FUNCTION_BLOCK FB_HMIManager EXTENDS FB_BaseGroupElement IMPLEMENTS ITF_HMIManager, ITF_HMIManagerConfigure
VAR
	(*	Inicjalizacja		*)
	bInitializeCycle			: BOOL;
	bInitDone					: BOOL;
	(*	Konfiguracja		*)
	itfHMIConfigure			: ITF_HMIConfigure;		//moduł konfiguracji
	(*	Menu główne	*)
	itfMainMenu				: ITF_HMIEMenu;
	iNumberOfButtonMainMenu	: INT;
	(*	Obsługa zmiany strony	*)
	arrChangePageSupport	: ARRAY [0..GVL_HMIEConstans.MAX_NUMBER_OF_BUTTON_IN_MENU] OF ITF_ChangePageSupport;
	(*	Dana wspólne dla całego systemu	*)
	refstData				: REFERENCE TO ST_HMIManager;
END_VAR

IF (NOT THIS^.bInitializeCycle) THEN
	THIS^.bInitializeCycle		:= TRUE;
	THIS^.bInitDone				:= THIS^.InitializeCycle ();
ELSIF (THIS^.bInitDone) THEN
	THIS^.ExecuteCycle ();
END_IF

(*			
	RafalOS
	Rafał Osajda		13.11.2025		TC 4024.66
	Dodawanie elementów wywoływane z konfiguracji 
*)
METHOD PUBLIC AddElementFromConfiguration : BOOL
VAR_INPUT
	itfElements		: ITF_BaseTopElement_HMI;
END_VAR
END_METHOD

(*			
	RafalOS
	Rafał Osajda		29.10.2025		TC 4024.66
	Dodawanie intefejsu konfiguracji
*)
METHOD PUBLIC AddModulConfigure : BOOL
VAR_INPUT
	fbHMIConfigure			: ITF_HMIConfigure;
END_VAR
THIS^.itfHMIConfigure		:= fbHMIConfigure;
END_METHOD

(*			
	RafalOS
	Rafał Osajda		10.11.2025		TC 4024.66
	Główna metoda sterujaca wyświetlaniem dsanych na HMI
*)
METHOD PUBLIC ExecuteCycle
(*
	(* Testowanie MenuGlownego	*)
THIS^.itfMainMenu.Testing ();

	(*	Aktualizacja zmiennych przy zmianie strony	*)
IF (THIS^.itfMainMenu.IsChangePage ()) THEN
	THIS^.refstData.iNUmberOfActivePage	:= THIS^.itfMainMenu.GetNumberOfActriveScreen ();
	
END_IF

	(*	Odświerzenia strrony 	*)
IF (THIS^.arrChangePageSupport [THIS^.refstData.iNUmberOfActivePage] <> 0) THEN
	THIS^.arrChangePageSupport [THIS^.refstData.iNUmberOfActivePage].PreparePage ();
	//wyczyszczenie po ramce 
	//przygotowanie ramki
END_IF
	(*	Skasowanie flagi zmiany strony	*)
THIS^.itfMainMenu.ResetChangePage ();
*)
END_METHOD

METHOD FB_init : BOOL
VAR_INPUT
	bInitRetains : BOOL; // if TRUE, the retain variables are initialized (warm start / cold start)
	bInCopyCode : BOOL;  // if TRUE, the instance afterwards gets moved into the copy code (online change)
END_VAR
THIS^.SetText (eLocation := E_BaseLocation.pl, wsDescription := "HMI Menadżer");
THIS^.SetText (eLocation := E_BaseLocation.en, wsDescription := "HMI Manager");
THIS^.SetText (eLocation := E_BaseLocation.de, wsDescription := "HMI Manager");
THIS^.SetName (stName := THIS^.GetTexts ());
END_METHOD

METHOD PRIVATE InitializeCycle : BOOL
VAR
	bResult					: BOOL;
	iI: INT;
END_VAR
bResult				:= TRUE;

bResult				:= bResult AND THIS^.itfHMIConfigure.Configure (fbHMIManager := THIS^);

InitializeCycle		:= bResult;
END_METHOD

METHOD PUBLIC SetActiveButtonMainMenuFromConfiguration : BOOL
VAR_INPUT
	iButton			: INT;	//numer przycisku od 0
	bValue			: BOOL;	//true aktywny może być tylko jeden w menu
END_VAR
THIS^.itfMainMenu.SetActiveButton (iButton := iButton, bIN := bValue);
END_METHOD

METHOD PUBLIC SetEnableButtonMainMenuFromConfiguration : BOOL
VAR_INPUT
	iButton			: INT;	//numer przycisku od 0
	bValue			: BOOL;	//true włączony
END_VAR
THIS^.itfMainMenu.SetEnableButton (iButton := iButton, bIN := bValue);
END_METHOD

METHOD PUBLIC SetVisibleButtonMainMenuFromConfiguration : BOOL
VAR_INPUT
	iButton			: INT;	//numer przycisku od 0
	bValue			: BOOL;	//true widoczny
END_VAR
THIS^.itfMainMenu.SetVisibleButton (iButton := iButton, bIN := bValue);
END_METHOD

METHOD PUBLIC STARE_AddMainMenu : BOOL
VAR_INPUT
	fbMenu				 : ITF_HMIEMenu;
END_VAR
THIS^.SetText (eLocation := E_BaseLocation.pl, wsDescription := "Menu główne");
THIS^.SetText (eLocation := E_BaseLocation.en, wsDescription := "Main menu");
THIS^.SetText (eLocation := E_BaseLocation.de, wsDescription := "Hauptmenü");
fbMenu.SetName (stName := THIS^.GetTexts ());
THIS^.AddControlElement (itfControlElement := fbMenu);

THIS^.itfMainMenu		:= fbMenu;
THIS^.itfMainMenu.LinkCommonData (stCommonData := THIS^.refstCommonData);
END_METHOD

END_FUNCTION_BLOCK

(* stored: Version 1.1.0.1
   POU FB_HMIManager: Id {a88b626b-1335-01ba-387a-b90d8f220c55}, SpecialFunc None
   Folder ITF_HMIManagerConfigure: Id {89138cc2-cb73-0422-3e5b-ed5c94136f56}
   Folder WiazanieModulow: Id {82c7cc63-7604-0b87-2d45-08cdf14b79c2}
   Method AddElementFromConfiguration: Id {c2b42e4c-e6c1-0e6a-3ae0-464a637c4e91}
   Method AddModulConfigure: Id {5f177fbc-999e-00c7-3b52-585090f74977}
   Method ExecuteCycle: Id {52b242f4-a20c-0dfc-3dbf-ca9f805176f3}
   Method FB_init: Id {85423e2b-17dc-0f54-335f-3500ae6327f4}
   Method InitializeCycle: Id {4e6e3c9a-8c44-48fc-b890-f0782f1c52b4}
   Method SetActiveButtonMainMenuFromConfiguration: Id {21ebb6b9-82ee-02ba-113e-377786737a20}
   Method SetEnableButtonMainMenuFromConfiguration: Id {39fad727-a855-013c-28c5-6e8efb5ac96d}
   Method SetVisibleButtonMainMenuFromConfiguration: Id {14e91481-d18f-0509-14ea-2677809820f7}
   Method STARE_AddMainMenu: Id {6015e53e-8f7a-0411-0f19-c77aa60698c6} *)
